FUNCTION_BLOCK EL3044
VAR
	_io : EL3xx4_Data;
	{attribute addProperty Name "WcState"}
	_wcState : WcStateInputToggle;
	{attribute addProperty Name "Info data"}
	_infoData : InfoDataAds;
END_VAR

PROPERTY IO : REFERENCE TO EL3xx4_Data
GET
IO REF= _io;
END_GET
END_PROPERTY

PROPERTY WcState : REFERENCE TO WcStateInputToggle
GET
WcState REF= _wcState;
END_GET
END_PROPERTY

END_FUNCTION_BLOCK

(* stored: Version 1.1.0.1, ProductVersion 3.1.4024.9
   POU EL3044: Id {209c0b23-903b-0e24-3083-04a976dcfdc7}, SpecialFunc None
   Property IO: Id {0c4e9361-4c32-031b-2ea0-be77c9391b57}
   Get Get: Id {282ac04b-ee1b-095c-199b-02ca4ec7c79c}
   Property WcState: Id {acaf52e4-2e21-0cb8-25a5-5342432d6987}
   Get Get: Id {786fb1af-85a9-007a-367e-28783eb6ce20} *)
